FUNCTION_BLOCK SystemTimeTick
VAR_INPUT
END_VAR
VAR_OUTPUT
END_VAR
VAR
	currentTicks : ULINT;
    timeMs : ULINT;
	timeS        : ULINT;  // seconds
    timeM        : ULINT;  // minutes
    timeH        : ULINT;  // hours
END_VAR

currentTicks := Tc2_System.F_GetSystemTime(); // returns system ticks

timeMs := currentTicks / 10000;   // convert to milliseconds (1 tick = 100ns)
timeS  := timeMs / 1000;                  // convert to seconds
timeM  := timeS / 60;                     // convert to minutes
timeH  := timeM / 60;                     // convert to hours

END_FUNCTION_BLOCK

(* stored: Version 1.1.0.1, ProductVersion 3.1.4024.13
   POU SystemTimeTick: Id {9c2a9c35-555a-4139-8bf0-7cebb4ce1fa5}, SpecialFunc None *)
